TYPE TcoGenericInterpolatorHwOutputs :
STRUCT
	qFromPlc AT %Q* : PLCTONC_NCICHANNEL_REF;
END_STRUCT
END_TYPE

(* stored: Version 1.1.0.1, ProductVersion 3.1.4024.12
   DUT TcoGenericInterpolatorHwOutputs: Id {9a6530dd-ac45-4b44-82d0-42c1c1cb6601} *)
